FUNCTION_BLOCK SENSOR_DB_SIM
  {SET_ATTRIBUTE(OpcUa, DEVICE.SENSOR)}
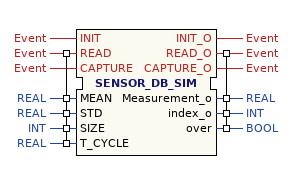
  EVENT_INPUT
    INIT;
    READ WITH MEAN, STD, SIZE, T_CYCLE;
    CAPTURE;
  END_EVENT
  EVENT_OUTPUT
    INIT_O;
    READ_O WITH Measurement_o, index_o, over;
    CAPTURE_O;
  END_EVENT
  VAR_INPUT
    MEAN : REAL; {SET_ATTRIBUTE(OpcUa, Variable)}
    STD : REAL; {SET_ATTRIBUTE(OpcUa, Variable)}
    SIZE : INT; {SET_ATTRIBUTE(OpcUa, Variable)}
    T_CYCLE : REAL; {SET_ATTRIBUTE(OpcUa, Variable)}
  END_VAR
  VAR_OUTPUT
    Measurement_o : REAL; {SET_ATTRIBUTE(OpcUa, Variable)}
    index_o : INT; {SET_ATTRIBUTE(OpcUa, Variable)}
    over : BOOL; {SET_ATTRIBUTE(OpcUa, Variable)}
  END_VAR
END_FUNCTION_BLOCK
